{attribute addProperty BoxType "EL6201-0000-0017"}
{attribute addProperty Id "Slave_23A_DI0BIT10.125177Slave_23A_DI1BIT10.125178Slave_23A_DI2BIT10.125179Slave_23A_DI3BIT10.125180Slave_23B_DI0BIT10.125181Slave_23B_DI1BIT10.125182Slave_23B_DI2BIT10.125183Slave_23B_DI3BIT10.125184"}
{attribute addProperty CRC "1699658775"}
{attribute addProperty SizeInBites "8"}
{attribute addProperty SizeInBytes "1"}
TYPE Slave_23_Inputs_654EBC17 :
STRUCT
	{attribute addProperty Name "Slave_23A_DI0"}
	Slave_23A_DI0 : BIT;
	{attribute addProperty Name "Slave_23A_DI1"}
	Slave_23A_DI1 : BIT;
	{attribute addProperty Name "Slave_23A_DI2"}
	Slave_23A_DI2 : BIT;
	{attribute addProperty Name "Slave_23A_DI3"}
	Slave_23A_DI3 : BIT;
	{attribute addProperty Name "Slave_23B_DI0"}
	Slave_23B_DI0 : BIT;
	{attribute addProperty Name "Slave_23B_DI1"}
	Slave_23B_DI1 : BIT;
	{attribute addProperty Name "Slave_23B_DI2"}
	Slave_23B_DI2 : BIT;
	{attribute addProperty Name "Slave_23B_DI3"}
	Slave_23B_DI3 : BIT;
END_STRUCT
END_TYPE

(* stored: Version 1.2.0.0, ProductVersion 3.1.4024.9
   DUT Slave_23_Inputs_654EBC17: Id {847da986-691e-403f-9d88-3cd5082abbe8} *)
